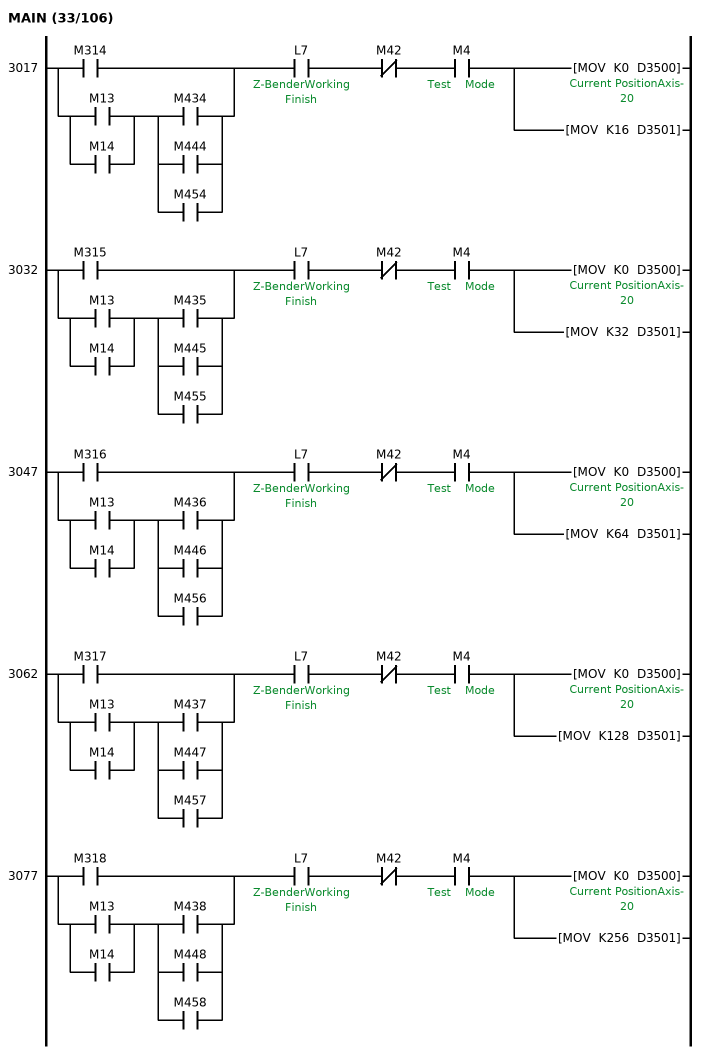
[picture p312: ladder of MAIN, rungs at steps 3017 to 3077]
3017  LD      M314
      LD      M13
      OR      M14
      LD      M434
      OR      M444
      OR      M454
      ANB
      ORB
      AND     L7  ; Z-BenderWorking Finish
      ANI     M42
      AND     M4  ; Test    Mode
      MOV     K0 D3500
      MOV     K16 D3501
3032  LD      M315
      LD      M13
      OR      M14
      LD      M435
      OR      M445
      OR      M455
      ANB
      ORB
      AND     L7  ; Z-BenderWorking Finish
      ANI     M42
      AND     M4  ; Test    Mode
      MOV     K0 D3500
      MOV     K32 D3501
3047  LD      M316
      LD      M13
      OR      M14
      LD      M436
      OR      M446
      OR      M456
      ANB
      ORB
      AND     L7  ; Z-BenderWorking Finish
      ANI     M42
      AND     M4  ; Test    Mode
      MOV     K0 D3500
      MOV     K64 D3501
3062  LD      M317
      LD      M13
      OR      M14
      LD      M437
      OR      M447
      OR      M457
      ANB
      ORB
      AND     L7  ; Z-BenderWorking Finish
      ANI     M42
      AND     M4  ; Test    Mode
      MOV     K0 D3500
      MOV     K128 D3501
3077  LD      M318
      LD      M13
      OR      M14
      LD      M438
      OR      M448
      OR      M458
      ANB
      ORB
      AND     L7  ; Z-BenderWorking Finish
      ANI     M42
      AND     M4  ; Test    Mode
      MOV     K0 D3500
      MOV     K256 D3501
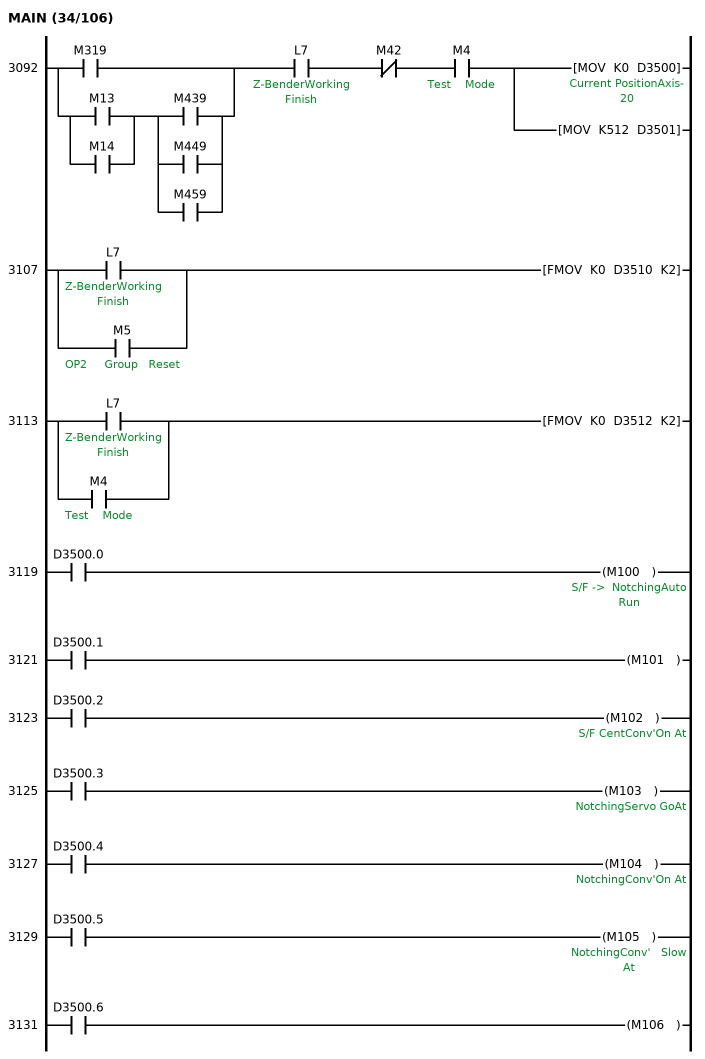
3092  LD      M319
      LD      M13
      OR      M14
      LD      M439
      OR      M449
      OR      M459
      ANB
      ORB
      AND     L7  ; Z-BenderWorking Finish
      ANI     M42
      AND     M4  ; Test    Mode
      MOV     K0 D3500
      MOV     K512 D3501
3107  LD      L7  ; Z-BenderWorking Finish
      OR      M5  ; OP2     Group   Reset
      FMOV    K0 D3510 K2
3113  LD      L7  ; Z-BenderWorking Finish
      OR      M4  ; Test    Mode
      FMOV    K0 D3512 K2
3119  LD      D3500.0
      OUT     M100  ; S/F ->  NotchingAuto Run
3121  LD      D3500.1
      OUT     M101
3123  LD      D3500.2
      OUT     M102  ; S/F CentConv'On At
3125  LD      D3500.3
      OUT     M103  ; NotchingServo GoAt
3127  LD      D3500.4
      OUT     M104  ; NotchingConv'On At
3129  LD      D3500.5
      OUT     M105  ; NotchingConv'   Slow At
3131  LD      D3500.6
      OUT     M106
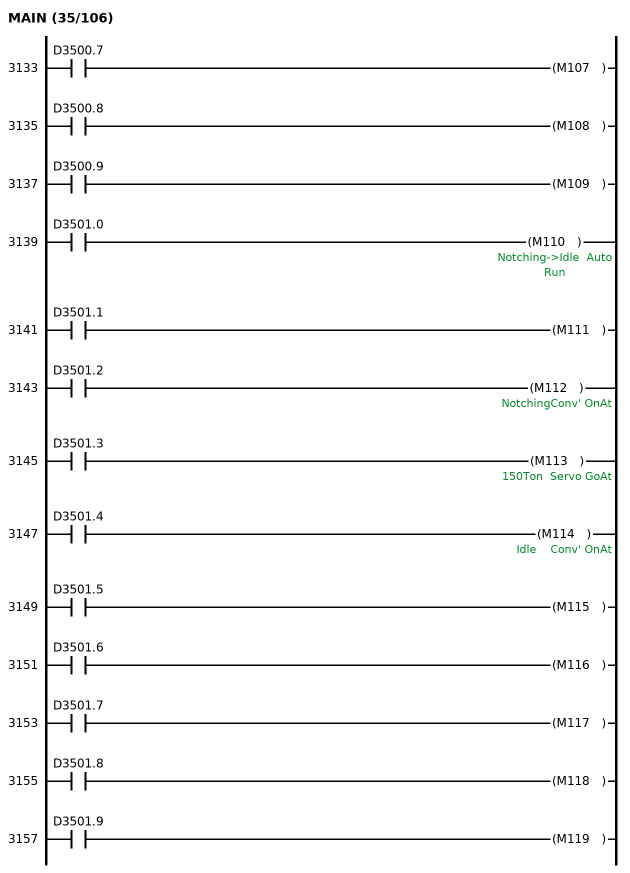
3133  LD      D3500.7
      OUT     M107
3135  LD      D3500.8
      OUT     M108
3137  LD      D3500.9
      OUT     M109
3139  LD      D3501.0
      OUT     M110  ; Notching->Idle  Auto Run
3141  LD      D3501.1
      OUT     M111
3143  LD      D3501.2
      OUT     M112  ; NotchingConv' OnAt
3145  LD      D3501.3
      OUT     M113  ; 150Ton  Servo GoAt
3147  LD      D3501.4
      OUT     M114  ; Idle    Conv' OnAt
3149  LD      D3501.5
      OUT     M115
3151  LD      D3501.6
      OUT     M116
3153  LD      D3501.7
      OUT     M117
3155  LD      D3501.8
      OUT     M118
3157  LD      D3501.9
      OUT     M119
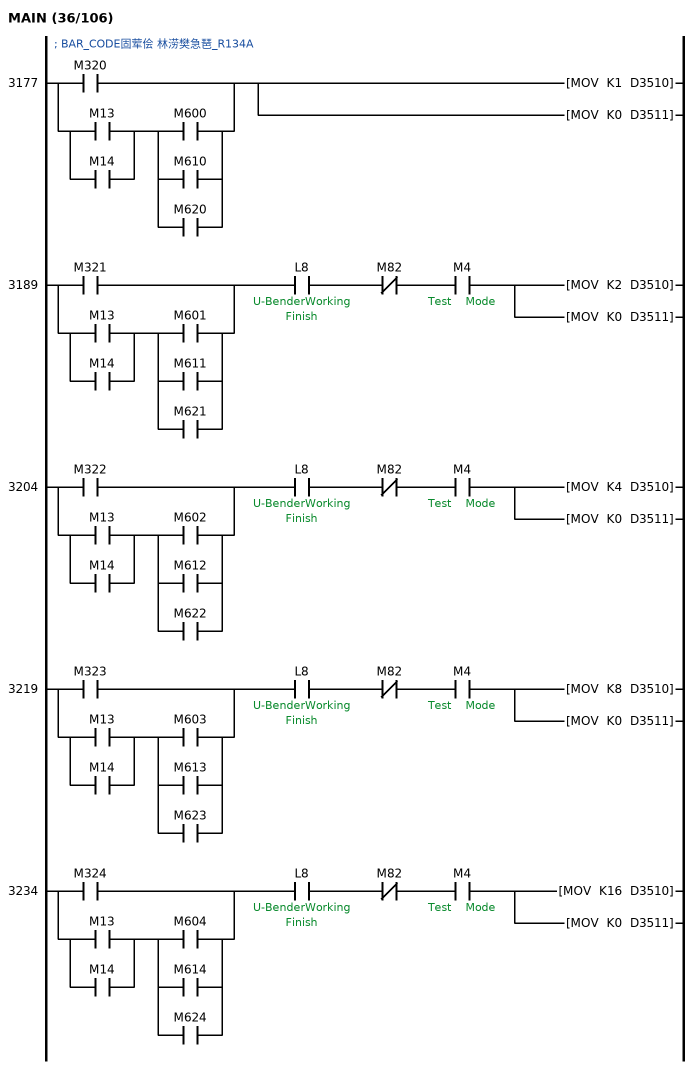
; BAR_CODE미사용 주입량선택_R134A
3177  LD      M320
      LD      M13
      OR      M14
      LD      M600
      OR      M610
      OR      M620
      ANB
      ORB
      MOV     K1 D3510
      MOV     K0 D3511
3189  LD      M321
      LD      M13
      OR      M14
      LD      M601
      OR      M611
      OR      M621
      ANB
      ORB
      AND     L8  ; U-BenderWorking Finish
      ANI     M82
      AND     M4  ; Test    Mode
      MOV     K2 D3510
      MOV     K0 D3511
3204  LD      M322
      LD      M13
      OR      M14
      LD      M602
      OR      M612
      OR      M622
      ANB
      ORB
      AND     L8  ; U-BenderWorking Finish
      ANI     M82
      AND     M4  ; Test    Mode
      MOV     K4 D3510
      MOV     K0 D3511
3219  LD      M323
      LD      M13
      OR      M14
      LD      M603
      OR      M613
      OR      M623
      ANB
      ORB
      AND     L8  ; U-BenderWorking Finish
      ANI     M82
      AND     M4  ; Test    Mode
      MOV     K8 D3510
      MOV     K0 D3511
3234  LD      M324
      LD      M13
      OR      M14
      LD      M604
      OR      M614
      OR      M624
      ANB
      ORB
      AND     L8  ; U-BenderWorking Finish
      ANI     M82
      AND     M4  ; Test    Mode
      MOV     K16 D3510
      MOV     K0 D3511
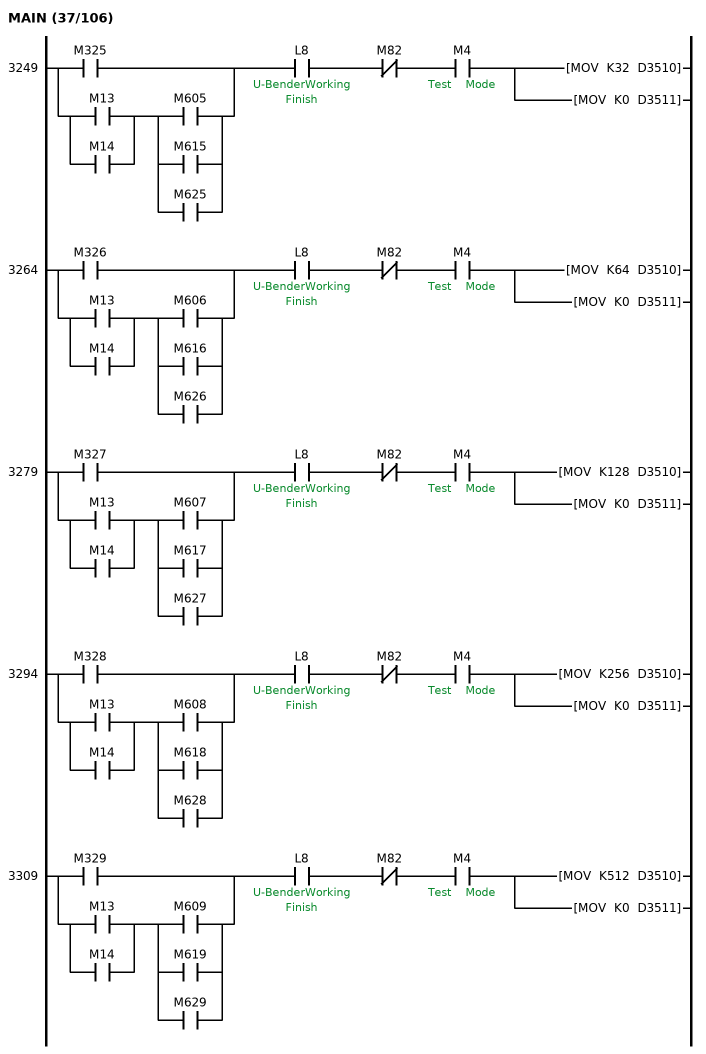
3249  LD      M325
      LD      M13
      OR      M14
      LD      M605
      OR      M615
      OR      M625
      ANB
      ORB
      AND     L8  ; U-BenderWorking Finish
      ANI     M82
      AND     M4  ; Test    Mode
      MOV     K32 D3510
      MOV     K0 D3511
3264  LD      M326
      LD      M13
      OR      M14
      LD      M606
      OR      M616
      OR      M626
      ANB
      ORB
      AND     L8  ; U-BenderWorking Finish
      ANI     M82
      AND     M4  ; Test    Mode
      MOV     K64 D3510
      MOV     K0 D3511
3279  LD      M327
      LD      M13
      OR      M14
      LD      M607
      OR      M617
      OR      M627
      ANB
      ORB
      AND     L8  ; U-BenderWorking Finish
      ANI     M82
      AND     M4  ; Test    Mode
      MOV     K128 D3510
      MOV     K0 D3511
3294  LD      M328
      LD      M13
      OR      M14
      LD      M608
      OR      M618
      OR      M628
      ANB
      ORB
      AND     L8  ; U-BenderWorking Finish
      ANI     M82
      AND     M4  ; Test    Mode
      MOV     K256 D3510
      MOV     K0 D3511
3309  LD      M329
      LD      M13
      OR      M14
      LD      M609
      OR      M619
      OR      M629
      ANB
      ORB
      AND     L8  ; U-BenderWorking Finish
      ANI     M82
      AND     M4  ; Test    Mode
      MOV     K512 D3510
      MOV     K0 D3511
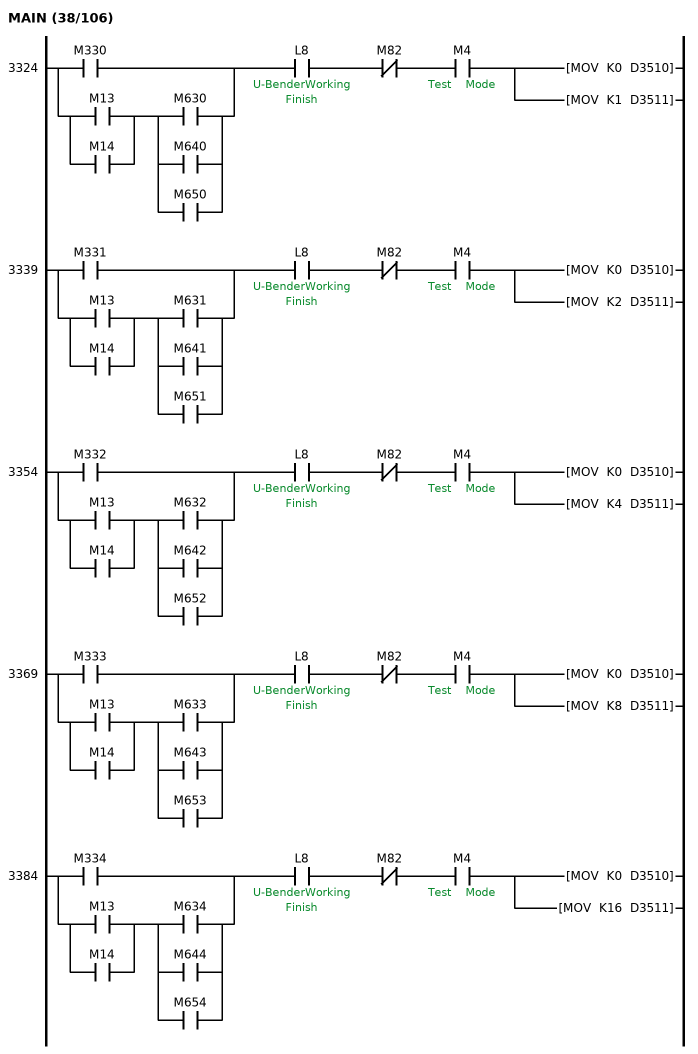
3324  LD      M330
      LD      M13
      OR      M14
      LD      M630
      OR      M640
      OR      M650
      ANB
      ORB
      AND     L8  ; U-BenderWorking Finish
      ANI     M82
      AND     M4  ; Test    Mode
      MOV     K0 D3510
      MOV     K1 D3511
3339  LD      M331
      LD      M13
      OR      M14
      LD      M631
      OR      M641
      OR      M651
      ANB
      ORB
      AND     L8  ; U-BenderWorking Finish
      ANI     M82
      AND     M4  ; Test    Mode
      MOV     K0 D3510
      MOV     K2 D3511
3354  LD      M332
      LD      M13
      OR      M14
      LD      M632
      OR      M642
      OR      M652
      ANB
      ORB
      AND     L8  ; U-BenderWorking Finish
      ANI     M82
      AND     M4  ; Test    Mode
      MOV     K0 D3510
      MOV     K4 D3511
3369  LD      M333
      LD      M13
      OR      M14
      LD      M633
      OR      M643
      OR      M653
      ANB
      ORB
      AND     L8  ; U-BenderWorking Finish
      ANI     M82
      AND     M4  ; Test    Mode
      MOV     K0 D3510
      MOV     K8 D3511
3384  LD      M334
      LD      M13
      OR      M14
      LD      M634
      OR      M644
      OR      M654
      ANB
      ORB
      AND     L8  ; U-BenderWorking Finish
      ANI     M82
      AND     M4  ; Test    Mode
      MOV     K0 D3510
      MOV     K16 D3511
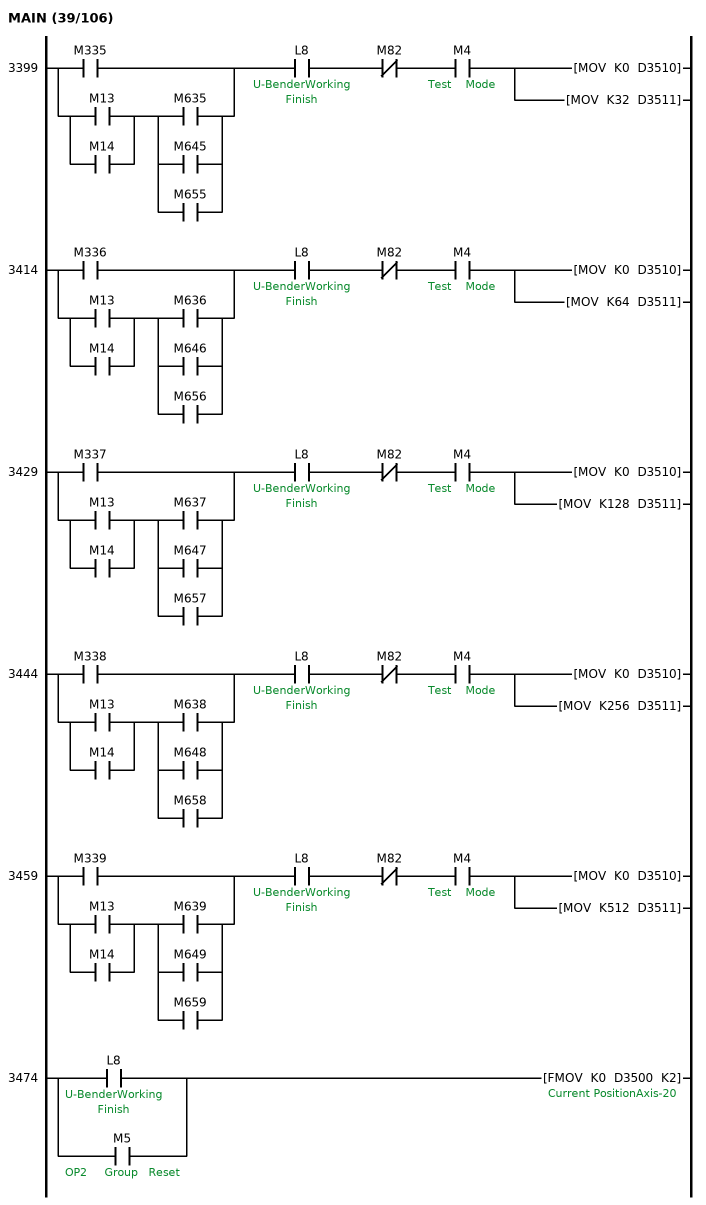
3399  LD      M335
      LD      M13
      OR      M14
      LD      M635
      OR      M645
      OR      M655
      ANB
      ORB
      AND     L8  ; U-BenderWorking Finish
      ANI     M82
      AND     M4  ; Test    Mode
      MOV     K0 D3510
      MOV     K32 D3511
3414  LD      M336
      LD      M13
      OR      M14
      LD      M636
      OR      M646
      OR      M656
      ANB
      ORB
      AND     L8  ; U-BenderWorking Finish
      ANI     M82
      AND     M4  ; Test    Mode
      MOV     K0 D3510
      MOV     K64 D3511
3429  LD      M337
      LD      M13
      OR      M14
      LD      M637
      OR      M647
      OR      M657
      ANB
      ORB
      AND     L8  ; U-BenderWorking Finish
      ANI     M82
      AND     M4  ; Test    Mode
      MOV     K0 D3510
      MOV     K128 D3511
3444  LD      M338
      LD      M13
      OR      M14
      LD      M638
      OR      M648
      OR      M658
      ANB
      ORB
      AND     L8  ; U-BenderWorking Finish
      ANI     M82
      AND     M4  ; Test    Mode
      MOV     K0 D3510
      MOV     K256 D3511
3459  LD      M339
      LD      M13
      OR      M14
      LD      M639
      OR      M649
      OR      M659
      ANB
      ORB
      AND     L8  ; U-BenderWorking Finish
      ANI     M82
      AND     M4  ; Test    Mode
      MOV     K0 D3510
      MOV     K512 D3511
3474  LD      L8  ; U-BenderWorking Finish
      OR      M5  ; OP2     Group   Reset
      FMOV    K0 D3500 K2
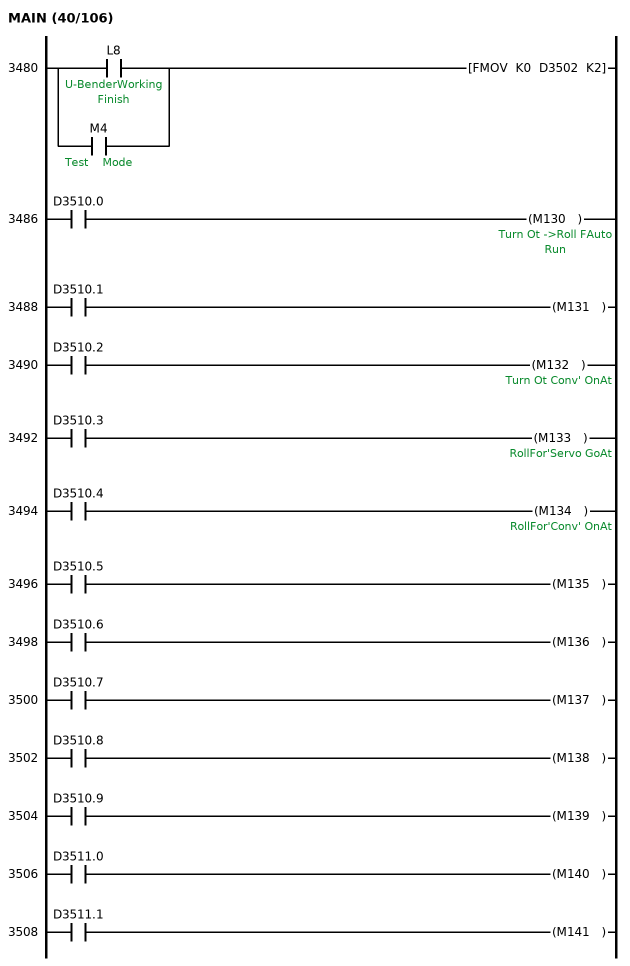
3480  LD      L8  ; U-BenderWorking Finish
      OR      M4  ; Test    Mode
      FMOV    K0 D3502 K2
3486  LD      D3510.0
      OUT     M130  ; Turn Ot ->Roll FAuto Run
3488  LD      D3510.1
      OUT     M131
3490  LD      D3510.2
      OUT     M132  ; Turn Ot Conv' OnAt
3492  LD      D3510.3
      OUT     M133  ; RollFor'Servo GoAt
3494  LD      D3510.4
      OUT     M134  ; RollFor'Conv' OnAt
3496  LD      D3510.5
      OUT     M135
3498  LD      D3510.6
      OUT     M136
3500  LD      D3510.7
      OUT     M137
3502  LD      D3510.8
      OUT     M138
3504  LD      D3510.9
      OUT     M139
3506  LD      D3511.0
      OUT     M140
3508  LD      D3511.1
      OUT     M141
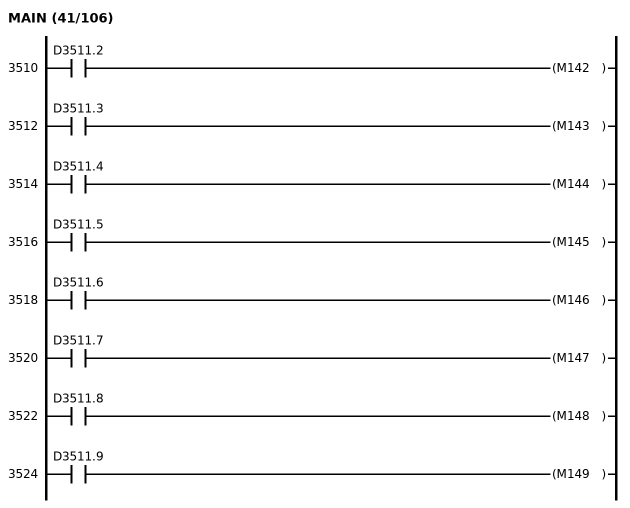
3510  LD      D3511.2
      OUT     M142
3512  LD      D3511.3
      OUT     M143
3514  LD      D3511.4
      OUT     M144
3516  LD      D3511.5
      OUT     M145
3518  LD      D3511.6
      OUT     M146
3520  LD      D3511.7
      OUT     M147
3522  LD      D3511.8
      OUT     M148
3524  LD      D3511.9
      OUT     M149
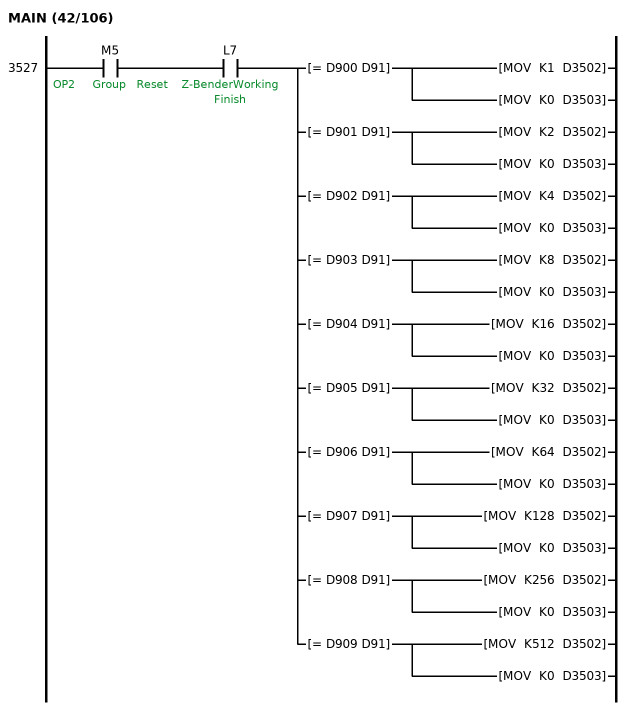
; 
3527  LD      M5  ; OP2     Group   Reset
      AND     L7  ; Z-BenderWorking Finish
      MPS
      AND=    D900 D91
      MOV     K1 D3502
      MOV     K0 D3503
      MRD
      AND=    D901 D91
      MOV     K2 D3502
      MOV     K0 D3503
      MRD
      AND=    D902 D91
      MOV     K4 D3502
      MOV     K0 D3503
      MRD
      AND=    D903 D91
      MOV     K8 D3502
      MOV     K0 D3503
      MRD
      AND=    D904 D91
      MOV     K16 D3502
      MOV     K0 D3503
      MRD
      AND=    D905 D91
      MOV     K32 D3502
      MOV     K0 D3503
      MRD
      AND=    D906 D91
      MOV     K64 D3502
      MOV     K0 D3503
      MRD
      AND=    D907 D91
      MOV     K128 D3502
      MOV     K0 D3503
      MRD
      AND=    D908 D91
      MOV     K256 D3502
      MOV     K0 D3503
      MPP
      AND=    D909 D91
      MOV     K512 D3502
      MOV     K0 D3503
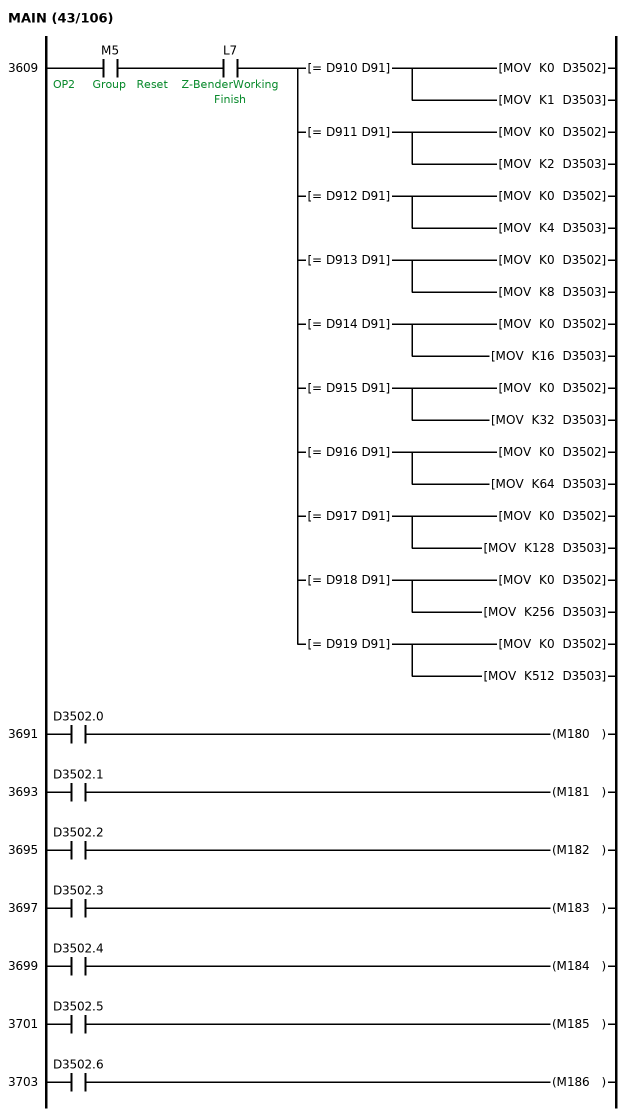
3609  LD      M5  ; OP2     Group   Reset
      AND     L7  ; Z-BenderWorking Finish
      MPS
      AND=    D910 D91
      MOV     K0 D3502
      MOV     K1 D3503
      MRD
      AND=    D911 D91
      MOV     K0 D3502
      MOV     K2 D3503
      MRD
      AND=    D912 D91
      MOV     K0 D3502
      MOV     K4 D3503
      MRD
      AND=    D913 D91
      MOV     K0 D3502
      MOV     K8 D3503
      MRD
      AND=    D914 D91
      MOV     K0 D3502
      MOV     K16 D3503
      MRD
      AND=    D915 D91
      MOV     K0 D3502
      MOV     K32 D3503
      MRD
      AND=    D916 D91
      MOV     K0 D3502
      MOV     K64 D3503
      MRD
      AND=    D917 D91
      MOV     K0 D3502
      MOV     K128 D3503
      MRD
      AND=    D918 D91
      MOV     K0 D3502
      MOV     K256 D3503
      MPP
      AND=    D919 D91
      MOV     K0 D3502
      MOV     K512 D3503
3691  LD      D3502.0
      OUT     M180
3693  LD      D3502.1
      OUT     M181
3695  LD      D3502.2
      OUT     M182
3697  LD      D3502.3
      OUT     M183
3699  LD      D3502.4
      OUT     M184
3701  LD      D3502.5
      OUT     M185
3703  LD      D3502.6
      OUT     M186
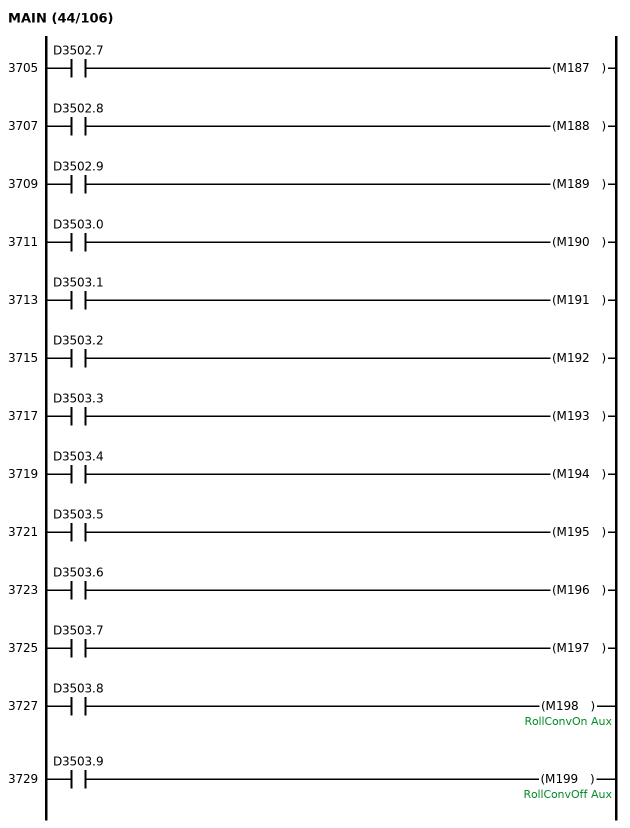
3705  LD      D3502.7
      OUT     M187
3707  LD      D3502.8
      OUT     M188
3709  LD      D3502.9
      OUT     M189
3711  LD      D3503.0
      OUT     M190
3713  LD      D3503.1
      OUT     M191
3715  LD      D3503.2
      OUT     M192
3717  LD      D3503.3
      OUT     M193
3719  LD      D3503.4
      OUT     M194
3721  LD      D3503.5
      OUT     M195
3723  LD      D3503.6
      OUT     M196
3725  LD      D3503.7
      OUT     M197
3727  LD      D3503.8
      OUT     M198  ; RollConvOn Aux
3729  LD      D3503.9
      OUT     M199  ; RollConvOff Aux
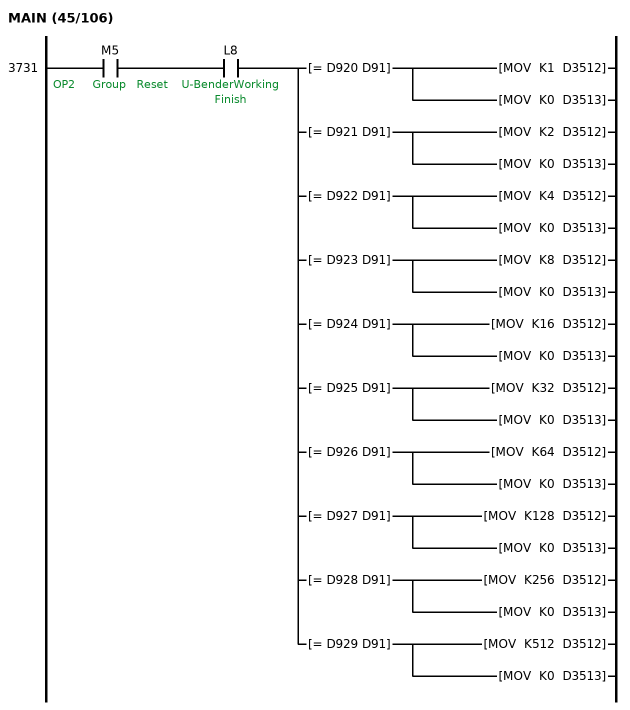
3731  LD      M5  ; OP2     Group   Reset
      AND     L8  ; U-BenderWorking Finish
      MPS
      AND=    D920 D91
      MOV     K1 D3512
      MOV     K0 D3513
      MRD
      AND=    D921 D91
      MOV     K2 D3512
      MOV     K0 D3513
      MRD
      AND=    D922 D91
      MOV     K4 D3512
      MOV     K0 D3513
      MRD
      AND=    D923 D91
      MOV     K8 D3512
      MOV     K0 D3513
      MRD
      AND=    D924 D91
      MOV     K16 D3512
      MOV     K0 D3513
      MRD
      AND=    D925 D91
      MOV     K32 D3512
      MOV     K0 D3513
      MRD
      AND=    D926 D91
      MOV     K64 D3512
      MOV     K0 D3513
      MRD
      AND=    D927 D91
      MOV     K128 D3512
      MOV     K0 D3513
      MRD
      AND=    D928 D91
      MOV     K256 D3512
      MOV     K0 D3513
      MPP
      AND=    D929 D91
      MOV     K512 D3512
      MOV     K0 D3513
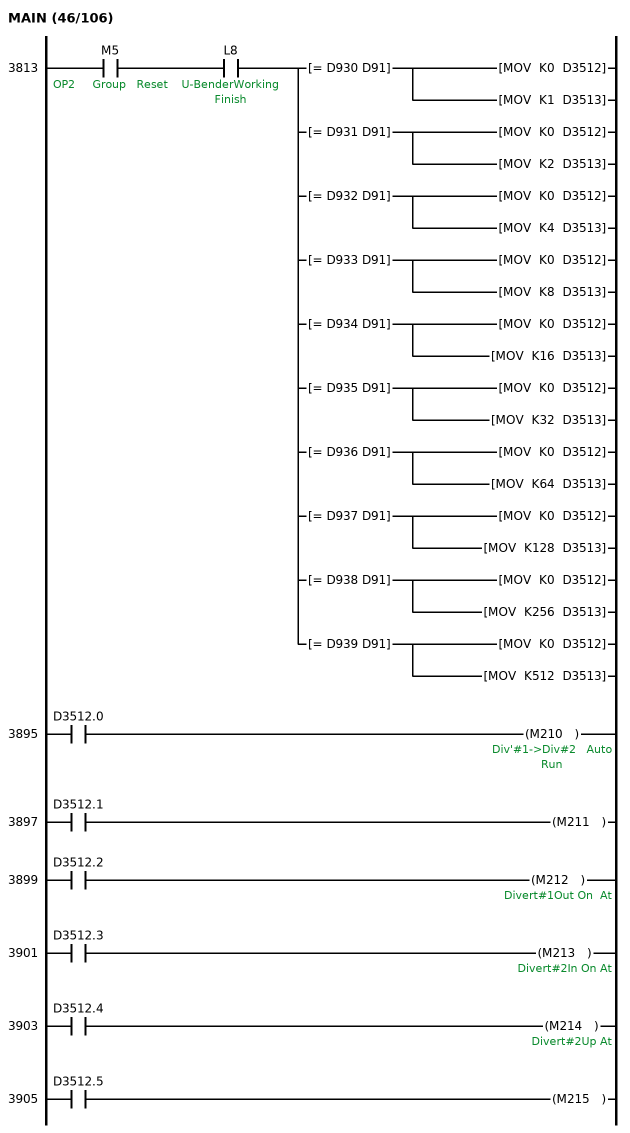
3813  LD      M5  ; OP2     Group   Reset
      AND     L8  ; U-BenderWorking Finish
      MPS
      AND=    D930 D91
      MOV     K0 D3512
      MOV     K1 D3513
      MRD
      AND=    D931 D91
      MOV     K0 D3512
      MOV     K2 D3513
      MRD
      AND=    D932 D91
      MOV     K0 D3512
      MOV     K4 D3513
      MRD
      AND=    D933 D91
      MOV     K0 D3512
      MOV     K8 D3513
      MRD
      AND=    D934 D91
      MOV     K0 D3512
      MOV     K16 D3513
      MRD
      AND=    D935 D91
      MOV     K0 D3512
      MOV     K32 D3513
      MRD
      AND=    D936 D91
      MOV     K0 D3512
      MOV     K64 D3513
      MRD
      AND=    D937 D91
      MOV     K0 D3512
      MOV     K128 D3513
      MRD
      AND=    D938 D91
      MOV     K0 D3512
      MOV     K256 D3513
      MPP
      AND=    D939 D91
      MOV     K0 D3512
      MOV     K512 D3513
3895  LD      D3512.0
      OUT     M210  ; Div'#1->Div#2   Auto Run
3897  LD      D3512.1
      OUT     M211
3899  LD      D3512.2
      OUT     M212  ; Divert#1Out On  At
3901  LD      D3512.3
      OUT     M213  ; Divert#2In On At
3903  LD      D3512.4
      OUT     M214  ; Divert#2Up At
3905  LD      D3512.5
      OUT     M215
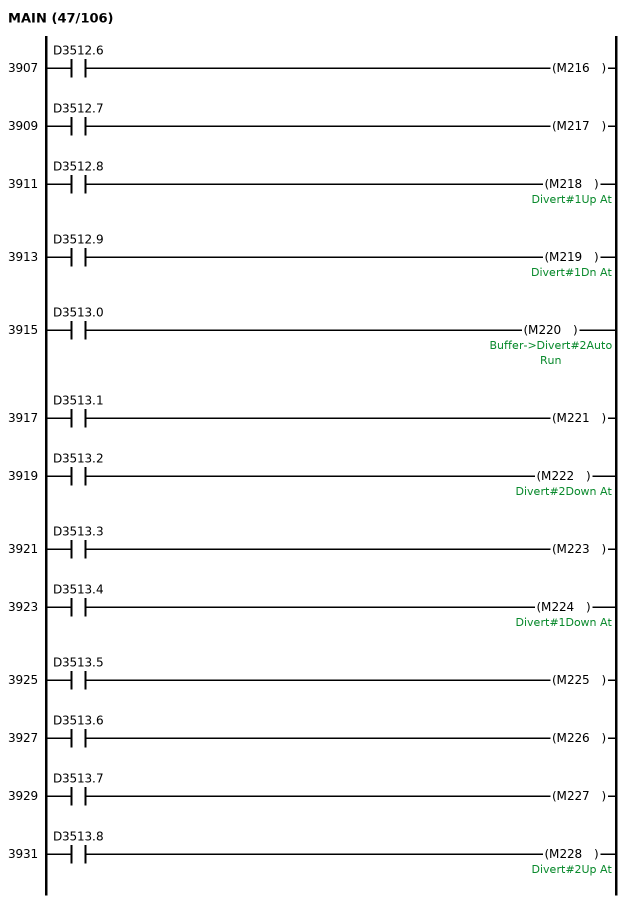
3907  LD      D3512.6
      OUT     M216
3909  LD      D3512.7
      OUT     M217
3911  LD      D3512.8
      OUT     M218  ; Divert#1Up At
3913  LD      D3512.9
      OUT     M219  ; Divert#1Dn At
3915  LD      D3513.0
      OUT     M220  ; Buffer->Divert#2Auto Run
3917  LD      D3513.1
      OUT     M221
3919  LD      D3513.2
      OUT     M222  ; Divert#2Down At
3921  LD      D3513.3
      OUT     M223
3923  LD      D3513.4
      OUT     M224  ; Divert#1Down At
3925  LD      D3513.5
      OUT     M225
3927  LD      D3513.6
      OUT     M226
3929  LD      D3513.7
      OUT     M227
3931  LD      D3513.8
      OUT     M228  ; Divert#2Up At
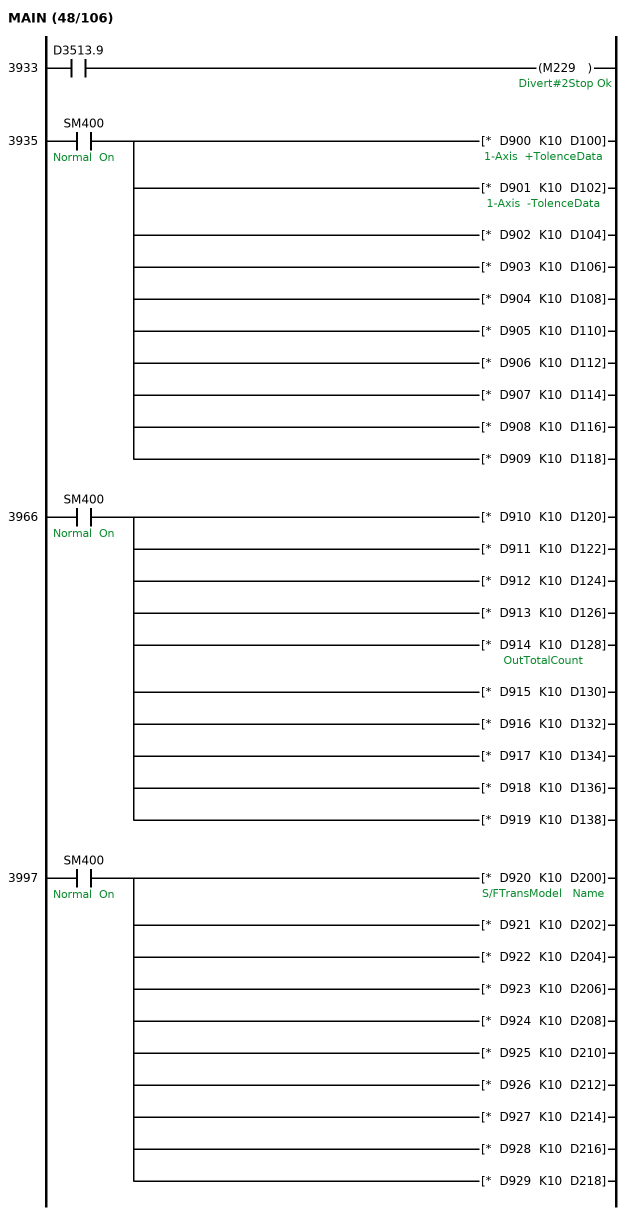
3933  LD      D3513.9
      OUT     M229  ; Divert#2Stop Ok
3935  LD      SM400  ; Normal  On
      *       D900 K10 D100  ; 1-Axis  +TolenceData
      *       D901 K10 D102  ; 1-Axis  -TolenceData
      *       D902 K10 D104
      *       D903 K10 D106
      *       D904 K10 D108
      *       D905 K10 D110
      *       D906 K10 D112
      *       D907 K10 D114
      *       D908 K10 D116
      *       D909 K10 D118
3966  LD      SM400  ; Normal  On
      *       D910 K10 D120
      *       D911 K10 D122
      *       D912 K10 D124
      *       D913 K10 D126
      *       D914 K10 D128  ; OutTotalCount
      *       D915 K10 D130
      *       D916 K10 D132
      *       D917 K10 D134
      *       D918 K10 D136
      *       D919 K10 D138
3997  LD      SM400  ; Normal  On
      *       D920 K10 D200  ; S/FTransModel   Name
      *       D921 K10 D202
      *       D922 K10 D204
      *       D923 K10 D206
      *       D924 K10 D208
      *       D925 K10 D210
      *       D926 K10 D212
      *       D927 K10 D214
      *       D928 K10 D216
      *       D929 K10 D218
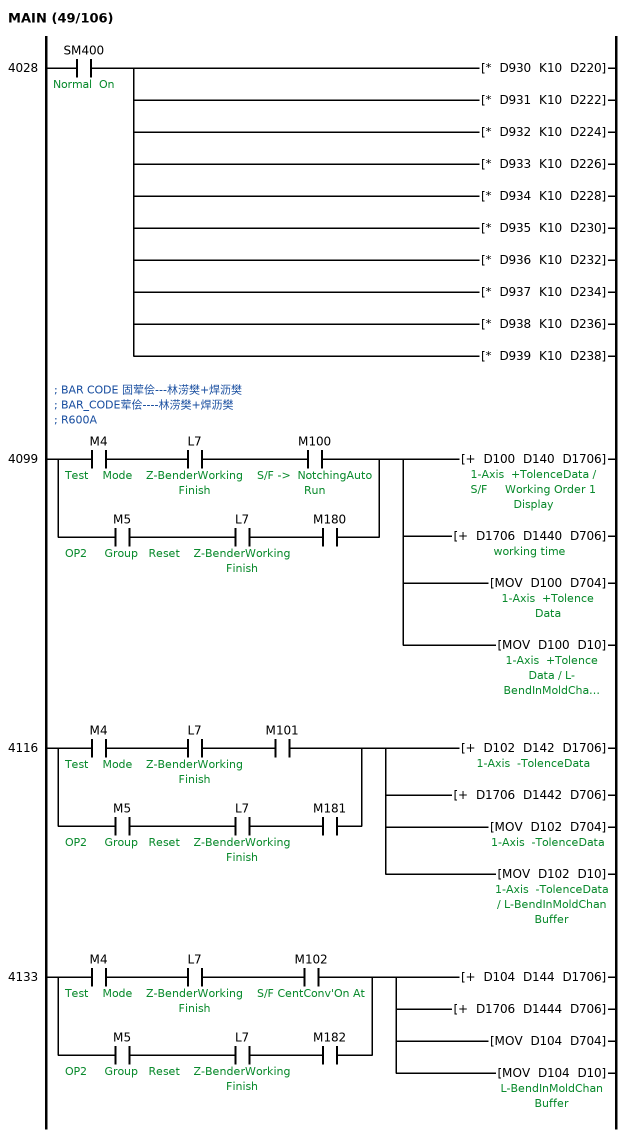
4028  LD      SM400  ; Normal  On
      *       D930 K10 D220
      *       D931 K10 D222
      *       D932 K10 D224
      *       D933 K10 D226
      *       D934 K10 D228
      *       D935 K10 D230
      *       D936 K10 D232
      *       D937 K10 D234
      *       D938 K10 D236
      *       D939 K10 D238
; BAR CODE 미사용---주입량+보정량
; BAR_CODE사용----주입량+보정량
; R600A
4099  LD      M4  ; Test    Mode
      AND     L7  ; Z-BenderWorking Finish
      AND     M100  ; S/F ->  NotchingAuto Run
      LD      M5  ; OP2     Group   Reset
      AND     L7  ; Z-BenderWorking Finish
      AND     M180
      ORB
      +       D100 D140 D1706  ; S/F     Working Order 1 Display
      +       D1706 D1440 D706  ; working time
      MOV     D100 D704
      MOV     D100 D10  ; L-BendInMoldChanBuffer
4116  LD      M4  ; Test    Mode
      AND     L7  ; Z-BenderWorking Finish
      AND     M101
      LD      M5  ; OP2     Group   Reset
      AND     L7  ; Z-BenderWorking Finish
      AND     M181
      ORB
      +       D102 D142 D1706
      +       D1706 D1442 D706
      MOV     D102 D704
      MOV     D102 D10
4133  LD      M4  ; Test    Mode
      AND     L7  ; Z-BenderWorking Finish
      AND     M102  ; S/F CentConv'On At
      LD      M5  ; OP2     Group   Reset
      AND     L7  ; Z-BenderWorking Finish
      AND     M182
      ORB
      +       D104 D144 D1706
      +       D1706 D1444 D706
      MOV     D104 D704
      MOV     D104 D10
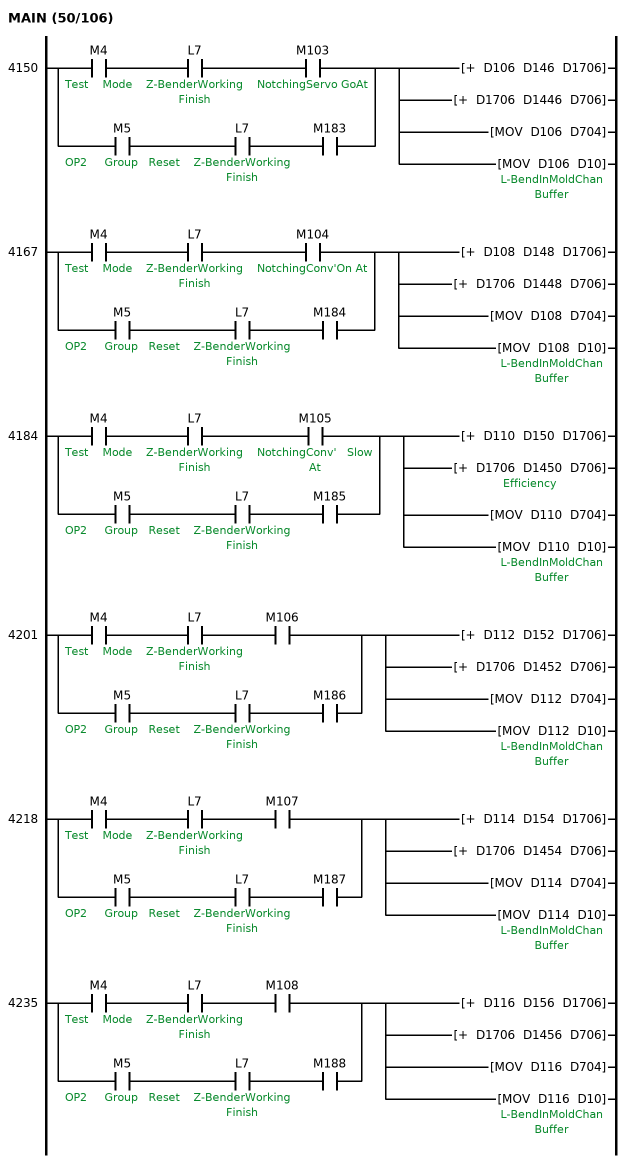
4150  LD      M4  ; Test    Mode
      AND     L7  ; Z-BenderWorking Finish
      AND     M103  ; NotchingServo GoAt
      LD      M5  ; OP2     Group   Reset
      AND     L7  ; Z-BenderWorking Finish
      AND     M183
      ORB
      +       D106 D146 D1706
      +       D1706 D1446 D706
      MOV     D106 D704
      MOV     D106 D10
4167  LD      M4  ; Test    Mode
      AND     L7  ; Z-BenderWorking Finish
      AND     M104  ; NotchingConv'On At
      LD      M5  ; OP2     Group   Reset
      AND     L7  ; Z-BenderWorking Finish
      AND     M184
      ORB
      +       D108 D148 D1706
      +       D1706 D1448 D706
      MOV     D108 D704
      MOV     D108 D10
4184  LD      M4  ; Test    Mode
      AND     L7  ; Z-BenderWorking Finish
      AND     M105  ; NotchingConv'   Slow At
      LD      M5  ; OP2     Group   Reset
      AND     L7  ; Z-BenderWorking Finish
      AND     M185
      ORB
      +       D110 D150 D1706
      +       D1706 D1450 D706  ; Efficiency
      MOV     D110 D704
      MOV     D110 D10
4201  LD      M4  ; Test    Mode
      AND     L7  ; Z-BenderWorking Finish
      AND     M106
      LD      M5  ; OP2     Group   Reset
      AND     L7  ; Z-BenderWorking Finish
      AND     M186
      ORB
      +       D112 D152 D1706
      +       D1706 D1452 D706
      MOV     D112 D704
      MOV     D112 D10
4218  LD      M4  ; Test    Mode
      AND     L7  ; Z-BenderWorking Finish
      AND     M107
      LD      M5  ; OP2     Group   Reset
      AND     L7  ; Z-BenderWorking Finish
      AND     M187
      ORB
      +       D114 D154 D1706
      +       D1706 D1454 D706
      MOV     D114 D704
      MOV     D114 D10
4235  LD      M4  ; Test    Mode
      AND     L7  ; Z-BenderWorking Finish
      AND     M108
      LD      M5  ; OP2     Group   Reset
      AND     L7  ; Z-BenderWorking Finish
      AND     M188
      ORB
      +       D116 D156 D1706
      +       D1706 D1456 D706
      MOV     D116 D704
      MOV     D116 D10
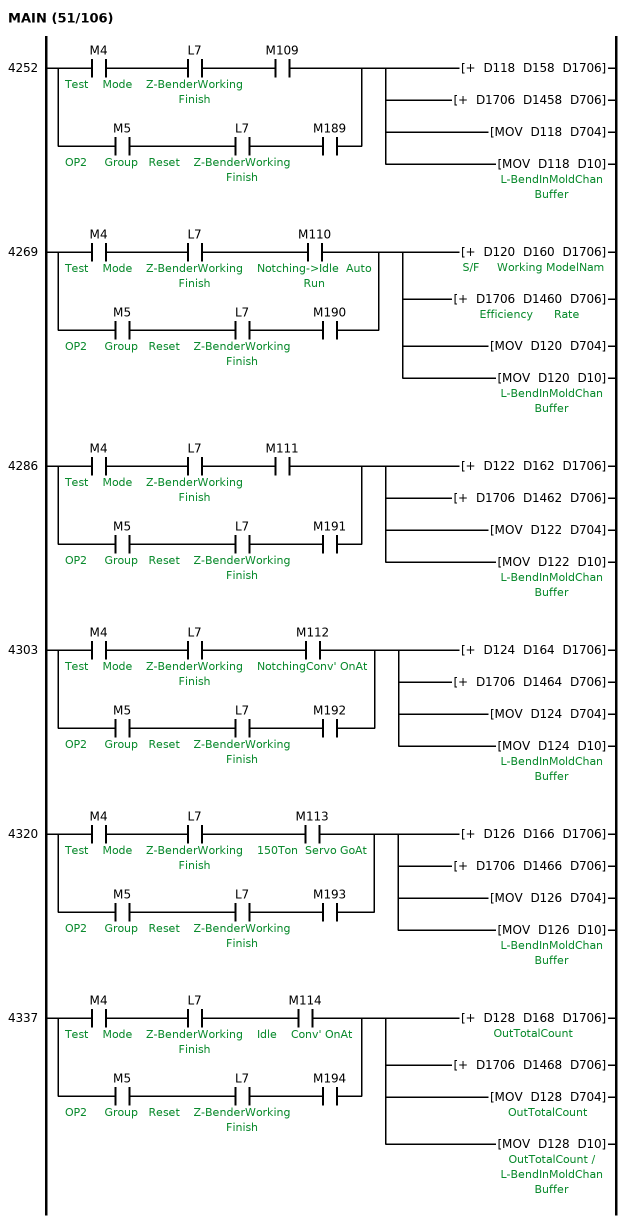
4252  LD      M4  ; Test    Mode
      AND     L7  ; Z-BenderWorking Finish
      AND     M109
      LD      M5  ; OP2     Group   Reset
      AND     L7  ; Z-BenderWorking Finish
      AND     M189
      ORB
      +       D118 D158 D1706
      +       D1706 D1458 D706
      MOV     D118 D704
      MOV     D118 D10
4269  LD      M4  ; Test    Mode
      AND     L7  ; Z-BenderWorking Finish
      AND     M110  ; Notching->Idle  Auto Run
      LD      M5  ; OP2     Group   Reset
      AND     L7  ; Z-BenderWorking Finish
      AND     M190
      ORB
      +       D120 D160 D1706  ; S/F     Working ModelNam
      +       D1706 D1460 D706  ; Efficiency      Rate
      MOV     D120 D704
      MOV     D120 D10
4286  LD      M4  ; Test    Mode
      AND     L7  ; Z-BenderWorking Finish
      AND     M111
      LD      M5  ; OP2     Group   Reset
      AND     L7  ; Z-BenderWorking Finish
      AND     M191
      ORB
      +       D122 D162 D1706
      +       D1706 D1462 D706
      MOV     D122 D704
      MOV     D122 D10
4303  LD      M4  ; Test    Mode
      AND     L7  ; Z-BenderWorking Finish
      AND     M112  ; NotchingConv' OnAt
      LD      M5  ; OP2     Group   Reset
      AND     L7  ; Z-BenderWorking Finish
      AND     M192
      ORB
      +       D124 D164 D1706
      +       D1706 D1464 D706
      MOV     D124 D704
      MOV     D124 D10
4320  LD      M4  ; Test    Mode
      AND     L7  ; Z-BenderWorking Finish
      AND     M113  ; 150Ton  Servo GoAt
      LD      M5  ; OP2     Group   Reset
      AND     L7  ; Z-BenderWorking Finish
      AND     M193
      ORB
      +       D126 D166 D1706
      +       D1706 D1466 D706
      MOV     D126 D704
      MOV     D126 D10
4337  LD      M4  ; Test    Mode
      AND     L7  ; Z-BenderWorking Finish
      AND     M114  ; Idle    Conv' OnAt
      LD      M5  ; OP2     Group   Reset
      AND     L7  ; Z-BenderWorking Finish
      AND     M194
      ORB
      +       D128 D168 D1706
      +       D1706 D1468 D706
      MOV     D128 D704
      MOV     D128 D10
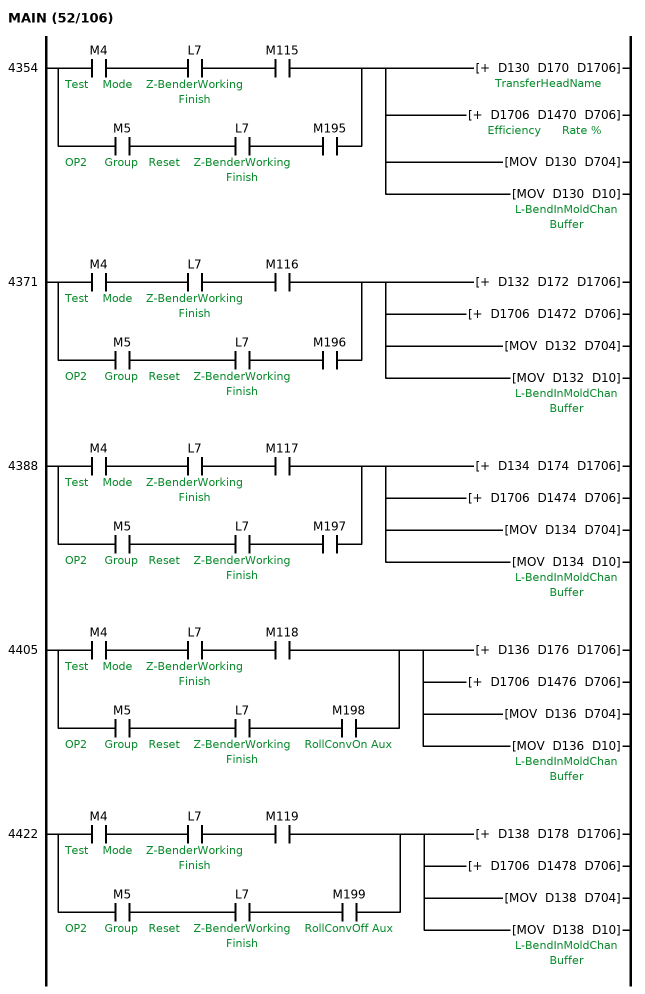
4354  LD      M4  ; Test    Mode
      AND     L7  ; Z-BenderWorking Finish
      AND     M115
      LD      M5  ; OP2     Group   Reset
      AND     L7  ; Z-BenderWorking Finish
      AND     M195
      ORB
      +       D130 D170 D1706  ; TransferHeadName
      +       D1706 D1470 D706  ; Efficiency      Rate %
      MOV     D130 D704
      MOV     D130 D10
4371  LD      M4  ; Test    Mode
      AND     L7  ; Z-BenderWorking Finish
      AND     M116
      LD      M5  ; OP2     Group   Reset
      AND     L7  ; Z-BenderWorking Finish
      AND     M196
      ORB
      +       D132 D172 D1706
      +       D1706 D1472 D706
      MOV     D132 D704
      MOV     D132 D10
4388  LD      M4  ; Test    Mode
      AND     L7  ; Z-BenderWorking Finish
      AND     M117
      LD      M5  ; OP2     Group   Reset
      AND     L7  ; Z-BenderWorking Finish
      AND     M197
      ORB
      +       D134 D174 D1706
      +       D1706 D1474 D706
      MOV     D134 D704
      MOV     D134 D10
4405  LD      M4  ; Test    Mode
      AND     L7  ; Z-BenderWorking Finish
      AND     M118
      LD      M5  ; OP2     Group   Reset
      AND     L7  ; Z-BenderWorking Finish
      AND     M198  ; RollConvOn Aux
      ORB
      +       D136 D176 D1706
      +       D1706 D1476 D706
      MOV     D136 D704
      MOV     D136 D10
4422  LD      M4  ; Test    Mode
      AND     L7  ; Z-BenderWorking Finish
      AND     M119
      LD      M5  ; OP2     Group   Reset
      AND     L7  ; Z-BenderWorking Finish
      AND     M199  ; RollConvOff Aux
      ORB
      +       D138 D178 D1706
      +       D1706 D1478 D706
      MOV     D138 D704
      MOV     D138 D10
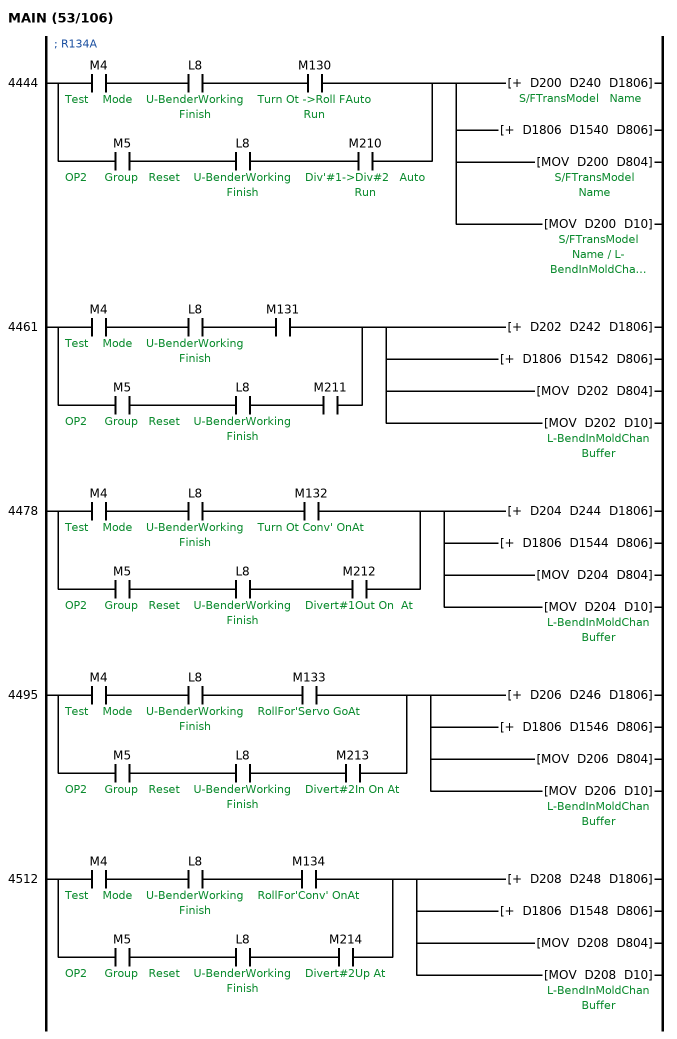
; R134A
4444  LD      M4  ; Test    Mode
      AND     L8  ; U-BenderWorking Finish
      AND     M130  ; Turn Ot ->Roll FAuto Run
      LD      M5  ; OP2     Group   Reset
      AND     L8  ; U-BenderWorking Finish
      AND     M210  ; Div'#1->Div#2   Auto Run
      ORB
      +       D200 D240 D1806
      +       D1806 D1540 D806
      MOV     D200 D804
      MOV     D200 D10
4461  LD      M4  ; Test    Mode
      AND     L8  ; U-BenderWorking Finish
      AND     M131
      LD      M5  ; OP2     Group   Reset
      AND     L8  ; U-BenderWorking Finish
      AND     M211
      ORB
      +       D202 D242 D1806
      +       D1806 D1542 D806
      MOV     D202 D804
      MOV     D202 D10
4478  LD      M4  ; Test    Mode
      AND     L8  ; U-BenderWorking Finish
      AND     M132  ; Turn Ot Conv' OnAt
      LD      M5  ; OP2     Group   Reset
      AND     L8  ; U-BenderWorking Finish
      AND     M212  ; Divert#1Out On  At
      ORB
      +       D204 D244 D1806
      +       D1806 D1544 D806
      MOV     D204 D804
      MOV     D204 D10
4495  LD      M4  ; Test    Mode
      AND     L8  ; U-BenderWorking Finish
      AND     M133  ; RollFor'Servo GoAt
      LD      M5  ; OP2     Group   Reset
      AND     L8  ; U-BenderWorking Finish
      AND     M213  ; Divert#2In On At
      ORB
      +       D206 D246 D1806
      +       D1806 D1546 D806
      MOV     D206 D804
      MOV     D206 D10
4512  LD      M4  ; Test    Mode
      AND     L8  ; U-BenderWorking Finish
      AND     M134  ; RollFor'Conv' OnAt
      LD      M5  ; OP2     Group   Reset
      AND     L8  ; U-BenderWorking Finish
      AND     M214  ; Divert#2Up At
      ORB
      +       D208 D248 D1806
      +       D1806 D1548 D806
      MOV     D208 D804
      MOV     D208 D10
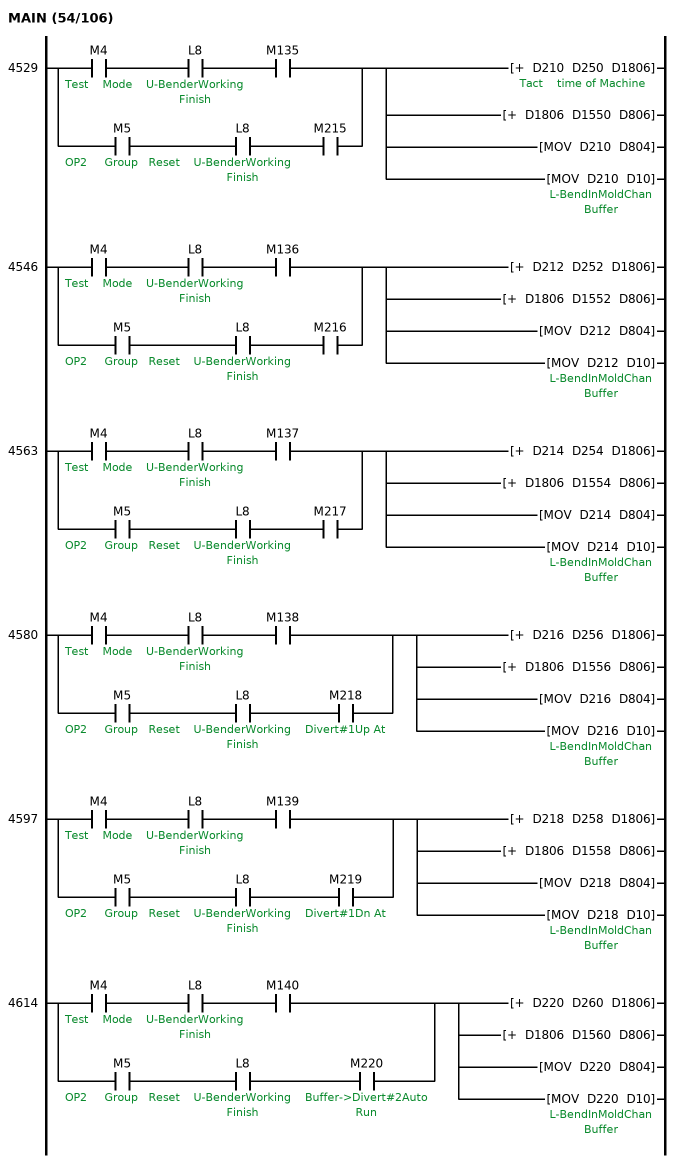
4529  LD      M4  ; Test    Mode
      AND     L8  ; U-BenderWorking Finish
      AND     M135
      LD      M5  ; OP2     Group   Reset
      AND     L8  ; U-BenderWorking Finish
      AND     M215
      ORB
      +       D210 D250 D1806  ; Tact    time of Machine
      +       D1806 D1550 D806
      MOV     D210 D804
      MOV     D210 D10
4546  LD      M4  ; Test    Mode
      AND     L8  ; U-BenderWorking Finish
      AND     M136
      LD      M5  ; OP2     Group   Reset
      AND     L8  ; U-BenderWorking Finish
      AND     M216
      ORB
      +       D212 D252 D1806
      +       D1806 D1552 D806
      MOV     D212 D804
      MOV     D212 D10
4563  LD      M4  ; Test    Mode
      AND     L8  ; U-BenderWorking Finish
      AND     M137
      LD      M5  ; OP2     Group   Reset
      AND     L8  ; U-BenderWorking Finish
      AND     M217
      ORB
      +       D214 D254 D1806
      +       D1806 D1554 D806
      MOV     D214 D804
      MOV     D214 D10
4580  LD      M4  ; Test    Mode
      AND     L8  ; U-BenderWorking Finish
      AND     M138
      LD      M5  ; OP2     Group   Reset
      AND     L8  ; U-BenderWorking Finish
      AND     M218  ; Divert#1Up At
      ORB
      +       D216 D256 D1806
      +       D1806 D1556 D806
      MOV     D216 D804
      MOV     D216 D10
4597  LD      M4  ; Test    Mode
      AND     L8  ; U-BenderWorking Finish
      AND     M139
      LD      M5  ; OP2     Group   Reset
      AND     L8  ; U-BenderWorking Finish
      AND     M219  ; Divert#1Dn At
      ORB
      +       D218 D258 D1806
      +       D1806 D1558 D806
      MOV     D218 D804
      MOV     D218 D10
4614  LD      M4  ; Test    Mode
      AND     L8  ; U-BenderWorking Finish
      AND     M140
      LD      M5  ; OP2     Group   Reset
      AND     L8  ; U-BenderWorking Finish
      AND     M220  ; Buffer->Divert#2Auto Run
      ORB
      +       D220 D260 D1806
      +       D1806 D1560 D806
      MOV     D220 D804
      MOV     D220 D10
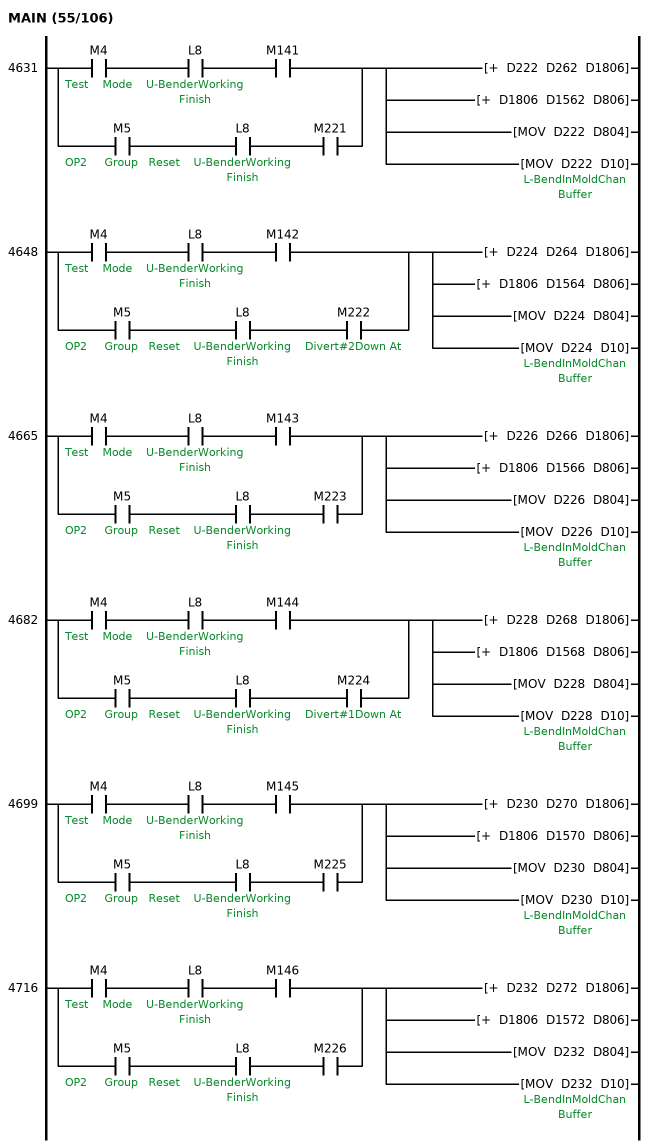
4631  LD      M4  ; Test    Mode
      AND     L8  ; U-BenderWorking Finish
      AND     M141
      LD      M5  ; OP2     Group   Reset
      AND     L8  ; U-BenderWorking Finish
      AND     M221
      ORB
      +       D222 D262 D1806
      +       D1806 D1562 D806
      MOV     D222 D804
      MOV     D222 D10
4648  LD      M4  ; Test    Mode
      AND     L8  ; U-BenderWorking Finish
      AND     M142
      LD      M5  ; OP2     Group   Reset
      AND     L8  ; U-BenderWorking Finish
      AND     M222  ; Divert#2Down At
      ORB
      +       D224 D264 D1806
      +       D1806 D1564 D806
      MOV     D224 D804
      MOV     D224 D10
4665  LD      M4  ; Test    Mode
      AND     L8  ; U-BenderWorking Finish
      AND     M143
      LD      M5  ; OP2     Group   Reset
      AND     L8  ; U-BenderWorking Finish
      AND     M223
      ORB
      +       D226 D266 D1806
      +       D1806 D1566 D806
      MOV     D226 D804
      MOV     D226 D10
4682  LD      M4  ; Test    Mode
      AND     L8  ; U-BenderWorking Finish
      AND     M144
      LD      M5  ; OP2     Group   Reset
      AND     L8  ; U-BenderWorking Finish
      AND     M224  ; Divert#1Down At
      ORB
      +       D228 D268 D1806
      +       D1806 D1568 D806
      MOV     D228 D804
      MOV     D228 D10
4699  LD      M4  ; Test    Mode
      AND     L8  ; U-BenderWorking Finish
      AND     M145
      LD      M5  ; OP2     Group   Reset
      AND     L8  ; U-BenderWorking Finish
      AND     M225
      ORB
      +       D230 D270 D1806
      +       D1806 D1570 D806
      MOV     D230 D804
      MOV     D230 D10
4716  LD      M4  ; Test    Mode
      AND     L8  ; U-BenderWorking Finish
      AND     M146
      LD      M5  ; OP2     Group   Reset
      AND     L8  ; U-BenderWorking Finish
      AND     M226
      ORB
      +       D232 D272 D1806
      +       D1806 D1572 D806
      MOV     D232 D804
      MOV     D232 D10
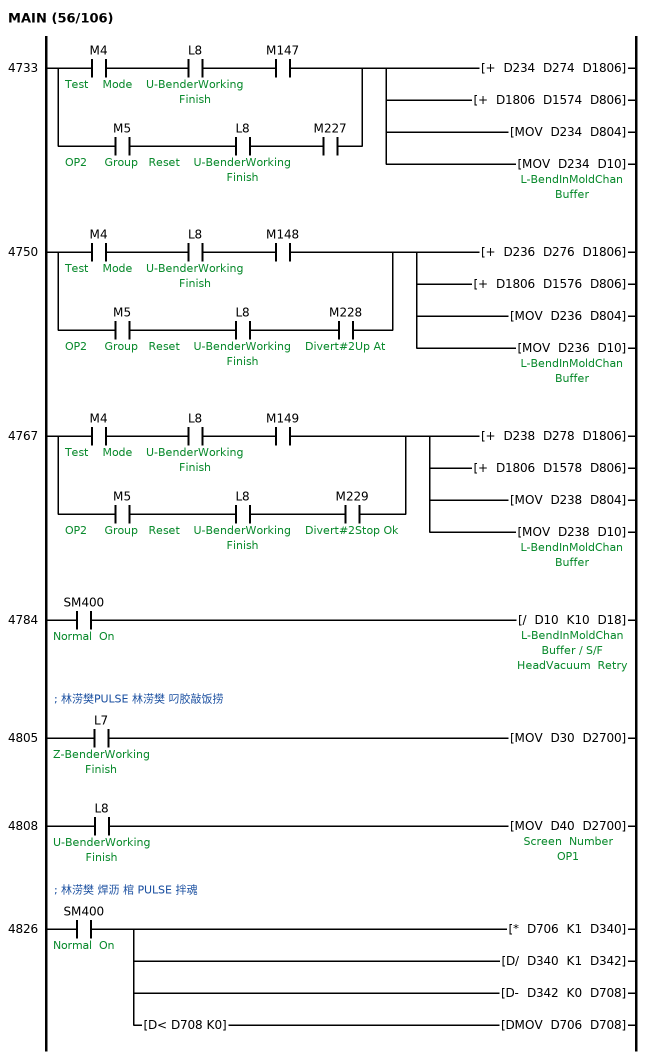
4733  LD      M4  ; Test    Mode
      AND     L8  ; U-BenderWorking Finish
      AND     M147
      LD      M5  ; OP2     Group   Reset
      AND     L8  ; U-BenderWorking Finish
      AND     M227
      ORB
      +       D234 D274 D1806
      +       D1806 D1574 D806
      MOV     D234 D804
      MOV     D234 D10
4750  LD      M4  ; Test    Mode
      AND     L8  ; U-BenderWorking Finish
      AND     M148
      LD      M5  ; OP2     Group   Reset
      AND     L8  ; U-BenderWorking Finish
      AND     M228  ; Divert#2Up At
      ORB
      +       D236 D276 D1806
      +       D1806 D1576 D806
      MOV     D236 D804
      MOV     D236 D10
4767  LD      M4  ; Test    Mode
      AND     L8  ; U-BenderWorking Finish
      AND     M149
      LD      M5  ; OP2     Group   Reset
      AND     L8  ; U-BenderWorking Finish
      AND     M229  ; Divert#2Stop Ok
      ORB
      +       D238 D278 D1806
      +       D1806 D1578 D806
      MOV     D238 D804
      MOV     D238 D10
4784  LD      SM400  ; Normal  On
      /       D10 K10 D18
; 주입량PULSE 주입량 디스플레이
4805  LD      L7  ; Z-BenderWorking Finish
      MOV     D30 D2700
4808  LD      L8  ; U-BenderWorking Finish
      MOV     D40 D2700
; 주입량 보정 및 PULSE 계산
4826  LD      SM400  ; Normal  On
      *       D706 K1 D340
      D/      D340 K1 D342
      D-      D342 K0 D708
      ANDD<   D708 K0
      DMOV    D706 D708
